{attribute 'linkalways'}
{attribute 'hide_all_locals'}
FUNCTION_BLOCK ValueTimeRead EXTENDS ValueBase IMPLEMENTS ValueRead
VAR
	thisValue : TIME;
END_VAR

{attribute 'call_after_global_init_slot' := '1'}
{attribute 'call_after_online_change_slot' := '1'}
METHOD PROTECTED GetThisAnyType
VAR_INPUT
END_VAR
thisAnyType := ToAnyType(thisValue);
END_METHOD

METHOD GetAsType : BOOL
VAR_INPUT
	destination : __SYSTEM.AnyType;
END_VAR
GetAsType := ConvertAnyType(thisAnyType, destination);
END_METHOD

METHOD GetAsString : T_MaxString
VAR_INPUT
END_VAR
GetAsString := TIME_TO_STRING(thisValue);
END_METHOD

METHOD Get : BOOL
VAR_INPUT
	destination : ANY;
END_VAR
Get := ConvertAnyType(thisAnyType, destination);
END_METHOD

METHOD FB_init : BOOL
VAR_INPUT
	bInitRetains : BOOL; // if TRUE, the retain variables are initialized (warm start / cold start)
	bInCopyCode : BOOL;  // if TRUE, the instance afterwards gets moved into the copy code (online change)
END_VAR
_ValueType := __SYSTEM.TYPE_CLASS.TYPE_TIME;
END_METHOD

{attribute 'monitoring' := 'call'}
PROPERTY Value : TIME
GET
Value := thisValue;
END_GET
END_PROPERTY

END_FUNCTION_BLOCK

(* stored: Version 1.1.0.1
   POU ValueTimeRead: Id {92d0234e-f8b8-4ae1-b42a-d11aaf36549c}, SpecialFunc None
   Method GetThisAnyType: Id {ff097832-fde4-4129-8eed-ea4065465cc4}
   Method GetAsType: Id {dee91efe-332c-4edb-8874-1f2b82837721}
   Method GetAsString: Id {6554e370-ae2b-4782-a8d3-2d8a75b4d5b6}
   Method Get: Id {0f3167b0-129f-4f2f-b2ea-dfa701abce6e}
   Method FB_init: Id {228dc079-8b14-4676-9a34-26b656725113}
   Property Value: Id {aa760726-6f48-4092-944b-7213d1ff5846}
   Get Get: Id {8ad68060-f808-4935-9c86-6ea9b1b83021} *)
